Staubli VAL3: AXIS7.dtx

public aio MbAI_a8Axispose = {link=ModbusSrv-0\Modbus-Word\MbAI_a8Axispose}
public aio MbAI_aCurPosH = {link=ModbusSrv-0\Modbus-Word\MbAI_aCurPosH}
public aio MbAI_aCurPosL = {link=ModbusSrv-0\Modbus-Word\MbAI_aCurPosL}
public aio MbAI_aUnused4 = {link=ModbusSrv-0\Modbus-Word\MbAI_aUnused4}
public aio MbAI_b8MotorErr = {link=ModbusSrv-0\Modbus-Word\MbAI_b8MotorError}
public aio MbAI_b8MotorPow = {link=ModbusSrv-0\Modbus-Word\MbAI_b8MotorPower}
public aio MbAI_bAxis7Reac = {link=ModbusSrv-0\Modbus-Word\MbAI_bAxis7Reached}
public aio MbAI_bAxis8Reac = {link=ModbusSrv-0\Modbus-Word\MbAI_bAxis8Reached}
public aio MbAI_bBackHome = {link=ModbusSrv-0\Modbus-Word\MbAI_bBackHome}
public aio MbAI_bDownLimit = {link=ModbusSrv-0\Modbus-Word\MbAI_bDownLimit}
public aio MbAI_bEndCycl = {link=ModbusSrv-0\Modbus-Word\MbAI_bEndCycl}
public aio MbAI_bHomeDone = {link=ModbusSrv-0\Modbus-Word\MbAI_bHomeDone}
public aio MbAI_bHomeLimit = {link=ModbusSrv-0\Modbus-Word\MbAI_bHomeLimit}
public aio MbAI_bIsHome = {link=ModbusSrv-0\Modbus-Word\MbAI_bIsHome}
public aio MbAI_bMotorErro = {link=ModbusSrv-0\Modbus-Word\MbAI_bMotorError}
public aio MbAI_bMotorPowe = {link=ModbusSrv-0\Modbus-Word\MbAI_bMotorPower}
public aio MbAI_bOutAlarm = {link=ModbusSrv-0\Modbus-Word\MbAI_bOutAlarm}
public aio MbAI_bPowerOn = {link=ModbusSrv-0\Modbus-Word\MbAI_bPowerOn}
public aio MbAI_bStartCycl = {link=ModbusSrv-0\Modbus-Word\MbAI_bStartCycl}
public aio MbAI_bUnused1 = {link=ModbusSrv-0\Modbus-Word\MbAI_bUnused1}
public aio MbAI_bUnused10 = {link=ModbusSrv-0\Modbus-Word\MbAI_bUnused10}
public aio MbAI_bUnused11 = {link=ModbusSrv-0\Modbus-Word\MbAI_bUnused11}
public aio MbAI_bUnused2 = {link=ModbusSrv-0\Modbus-Word\MbAI_bUnused2}
public aio MbAI_bUnused3 = {link=ModbusSrv-0\Modbus-Word\MbAI_bUnused3}
public aio MbAI_bUnused5 = {link=ModbusSrv-0\Modbus-Word\MbAI_bUnused5}
public aio MbAI_bUnused6 = {link=ModbusSrv-0\Modbus-Word\MbAI_bUnused6}
public aio MbAI_bUnused7 = {link=ModbusSrv-0\Modbus-Word\MbAI_bUnused7}
public aio MbAI_bUnused8 = {link=ModbusSrv-0\Modbus-Word\MbAI_bUnused8}
public aio MbAI_bUnused9 = {link=ModbusSrv-0\Modbus-Word\MbAI_bUnused9}
public aio MbAI_bUpLimit = {link=ModbusSrv-0\Modbus-Word\MbAI_bUpLimit}
public aio MbAO_aAxis7Puls = {link=ModbusSrv-0\Modbus-Word\MbAO_aAxis7Pulse}
public aio MbAO_aAxis8Puls = {link=ModbusSrv-0\Modbus-Word\MbAO_aAxis8Pulse}
public aio MbAO_aJogVelo = {link=ModbusSrv-0\Modbus-Word\MbAO_aJogVelo}
public aio MbAO_aJogVelo8 = {link=ModbusSrv-0\Modbus-Word\MbAO_aJogVelo8}
public aio MbAO_aMoveDis = {link=ModbusSrv-0\Modbus-Word\MbAO_aMoveDis}
public aio MbAO_aMoveDis8 = {link=ModbusSrv-0\Modbus-Word\MbAO_aMoveDis8}
public aio MbAO_aMovePosH = {link=ModbusSrv-0\Modbus-Word\MbAO_aMovePosH}
public aio MbAO_aMovePosH8 = {link=ModbusSrv-0\Modbus-Word\MbAO_aMovePosH8}
public aio MbAO_aMovePosL = {link=ModbusSrv-0\Modbus-Word\MbAO_aMovePosL}
public aio MbAO_aMovePosL8 = {link=ModbusSrv-0\Modbus-Word\MbAO_aMovePosL8}
public aio MbAO_aUnused10 = {link=ModbusSrv-0\Modbus-Word\MbAO_aUnused10}
public aio MbAO_aUnused11 = {link=ModbusSrv-0\Modbus-Word\MbAO_aUnused11}
public aio MbAO_aUnused6 = {link=ModbusSrv-0\Modbus-Word\MbAO_aUnused6}
public aio MbAO_aUnused7 = {link=ModbusSrv-0\Modbus-Word\MbAO_aUnused7}
public aio MbAO_aUnused8 = {link=ModbusSrv-0\Modbus-Word\MbAO_aUnused8}
public aio MbAO_aUnused9 = {link=ModbusSrv-0\Modbus-Word\MbAO_aUnused9}
public aio MbAO_aVelocity = {link=ModbusSrv-0\Modbus-Word\MbAO_aVelocity}
public aio MbAO_aVelocity8 = {link=ModbusSrv-0\Modbus-Word\MbAO_aVelocity8}
public aio MbAO_b7Axis = {link=ModbusSrv-0\Modbus-Word\MbAO_b7Axis}
public aio MbAO_b8Axis = {link=ModbusSrv-0\Modbus-Word\MbAO_b8Axis}
public aio MbAO_bAxis7Dire = {link=ModbusSrv-0\Modbus-Word\MbAO_bAxis7Direction}
public aio MbAO_bAxis7Home = {link=ModbusSrv-0\Modbus-Word\MbAO_bAxis7Home}
public aio MbAO_bAxis8Dire = {link=ModbusSrv-0\Modbus-Word\MbAO_bAxis8Direction}
public aio MbAO_bMoveDir = {link=ModbusSrv-0\Modbus-Word\MbAO_bMoveDir}
public aio MbAO_bMoveDirM = {link=ModbusSrv-0\Modbus-Word\MbAO_bMoveDirM}
public aio MbAO_bMovePos8 = {link=ModbusSrv-0\Modbus-Word\MbAO_bMovePos8}
public aio MbAO_bMoveToPos = {link=ModbusSrv-0\Modbus-Word\MbAO_bMoveToPos}
public aio MbAO_bRecordPos = {link=ModbusSrv-0\Modbus-Word\MbAO_bRecordPos}
public aio MbAO_bResetErr = {link=ModbusSrv-0\Modbus-Word\MbAO_bResetErr}
public aio MbAO_bStopMotor = {link=ModbusSrv-0\Modbus-Word\MbAO_bStopMotor}
public aio MbAO_bUnused1 = {link=ModbusSrv-0\Modbus-Word\MbAO_bUnused1}
public aio MbAO_bUnused2 = {link=ModbusSrv-0\Modbus-Word\MbAO_bUnused2}
public aio MbAO_bUnused3 = {link=ModbusSrv-0\Modbus-Word\MbAO_bUnused3}
public aio MbAO_bUnused4 = {link=ModbusSrv-0\Modbus-Word\MbAO_bUnused4}
public aio MbAO_bUnused5 = {link=ModbusSrv-0\Modbus-Word\MbAO_bUnused5}
public bool bAxisRun
num i = 6
public num nSaveaxis[7]
  [0] = 17569
  [1] = 17753
  [2] = 17775
  [3] = 17555
  [4] = 17803
  [5] = 17805
  [6] = 17722
public num nSaveaxis1[7]
  [0] = 36925
  [1] = 31321
  [2] = 60066
  [3] = 25553
  [4] = 27683
  [5] = 48927
  [6] = 32566
public num nVelocity[7]
  [0] = 8
  [1] = 8
  [2] = 8
  [3] = 8
  [4] = 8
  [5] = 8
  [6] = 8
string l_sItem = "PStart"
public string sItems
public string sSaveaxis[7]
  [0] = "workPos"
  [1] = "p1"
  [2] = "PStart"
  [3] = "P_001"
  [4] = "P_002"
  [5] = "PEnd"
  [6] = "PSychro"
